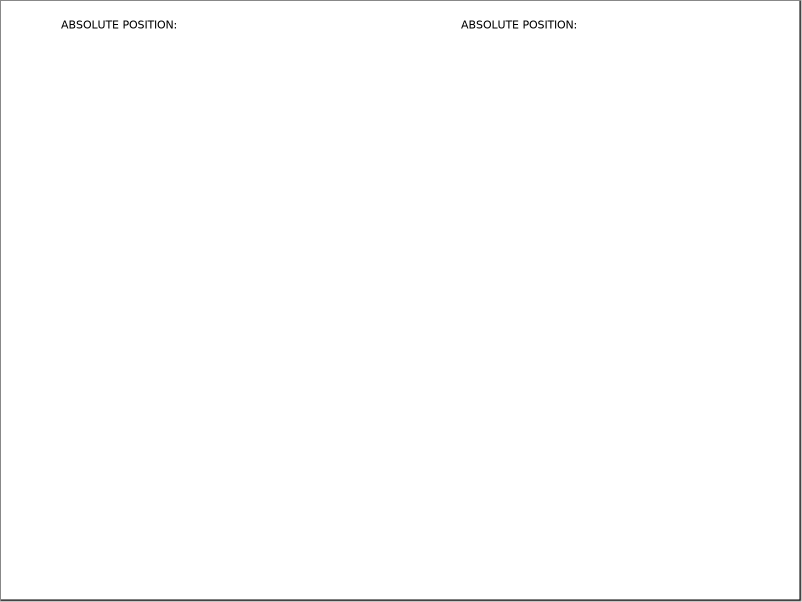
VISUALIZATION F07_Write_Parameter  // 802x602
    Rectangle (0,0 800x600)
    Label (10,10 170x30), "ABSOLUTE POSITION:"
    Label (410,10 170x30), "ABSOLUTE POSITION:"
END_VISUALIZATION

(* stored: Version 1.1.0.1, ProductVersion 3.1.4022.7
   Visu F07_Write_Parameter: Id {b5b68905-0238-4aea-83e2-af1b7068deba} *)
